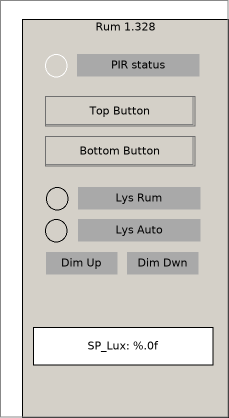
VISUALIZATION Visualization_1_328  // 229x418
    RoundedRectangle (22,19 207x399), "Rum 1.328"
    Rectangle (33,327 180x38), "SP_Lux: %.0f", text variable: P_Rum_1_328.fbLys.fbLightCtrl.fLuxZone1
    Button (45,96 150x30), "Top Button"
        tap P_Rum_1_328.bTopButtonZone1_Visu
    Button (45,136 150x30), "Bottom Button"
        tap P_Rum_1_328.bBottomButtonZone1_Visu
    Ellipse (46,187 22x23), colour toggle: P_Rum_1_328.fbLys.fbLightCtrl.bOnZone1
    Rectangle (78,187 122x22), "Lys Rum"
    Rectangle (46,252 71x22), "Dim Up", colour toggle: P_Rum_1_328.fbLys.fbLightCtrl.bDimUp
    Rectangle (127,252 71x22), "Dim Dwn", colour toggle: P_Rum_1_328.fbLys.fbLightCtrl.bDimDwn
    Ellipse (45,219 22x23), colour toggle: P_Rum_1_328.fbLightCtrl.bAutoZone1
    Rectangle (78,219 122x22), "Lys Auto"
    Ellipse (45,54 22x23), colour toggle: P_Rum_1_328.fbLys.fbLightCtrl.bPIR
    Rectangle (77,54 122x22), "PIR status"
END_VISUALIZATION

(* stored: Version 1.1.0.1
   Visu Visualization_1_328: Id {e9877f76-7ece-437d-bfd3-707b503b84f5} *)
